# EPICS substitutions: apps/harp_genericApp/Db/moeller_target.substitutions
file "db/motor.db" {
pattern {     motor_name, card, slot, srev, urev, direction, velo, accl }
        { moeller_target,    1,    0, 2000, 0.2,       Neg,  0.5, 0.1 }

}
